{region '#Template'}
	{attribute 'Version' := '1.2.2.0'}
	{attribute 'Tags' := '"LCID": "1031", "Text": "AC, Aggregates, Cooler, Temperature, Controller"'}
	{attribute 'Tags' := '"LCID": "1033", "Text": "AC, Aggregates, Cooler, Temperature, Controller"'}
	{attribute 'Using' := '"Type": "Template", "URI": "BA2_Param"'}
	{attribute 'Using' := '"Type": "Template", "URI": "EC_AMEV"'}
	{attribute 'Description' := '"LCID": "1031", "Text": "Kühler Zuluft Regler Temperatur"'}
	{attribute 'Description' := '"LCID": "1033", "Text": "Cooler Supply air controller temperature"'}
{endregion}
FUNCTION_BLOCK FB_BA_AC_ColTSuACtrl EXTENDS FB_BA_View
VAR_INPUT
	bEn						: BOOL;
	fSpTSuA					: REAL;// Sollwert Temperatur kühlen // Setpoint temperature cooling
	fTSuA					: REAL;// Zuluft Temperatur // Supply air temperature
	bSync					: BOOL;
	fSync					: REAL;
END_VAR
VAR_OUTPUT
	fY              		: REAL;
	bIsActive				: BOOL;	//	active sequence controller
	bOpState				: BOOL;	//	Release sequence link, sequence control is active	
END_VAR
VAR_INPUT CONSTANT
	Ctrl					: FB_BA_LoopSeq;
END_VAR

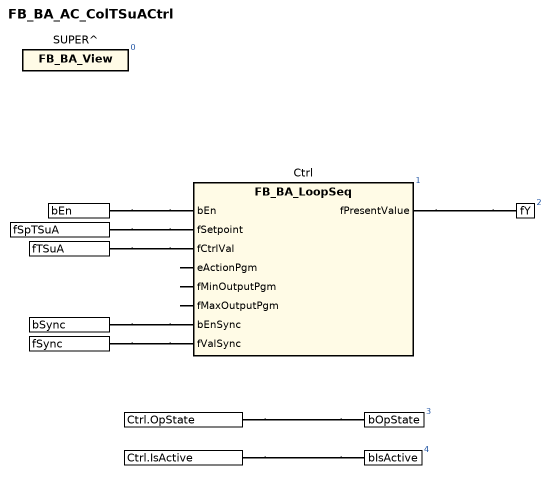
SUPER^(); // FB_BA_View
Ctrl(bEn := bEn, fSetpoint := fSpTSuA, fCtrlVal := fTSuA, bEnSync := bSync, fValSync := fSync); // FB_BA_LoopSeq
fY := Ctrl.fPresentValue;
bOpState := Ctrl.OpState;
bIsActive := Ctrl.IsActive;

METHOD FB_init : BOOL
VAR_INPUT
	bInitRetains : BOOL; // if TRUE, the retain variables are initialized (warm start / cold start)
	bInCopyCode : BOOL;  // if TRUE, the instance afterwards gets moved into the copy code (online change)
END_VAR
Ctrl.iParent						:= THIS^;
Ctrl.iLabel							:= LblCmpAC.Cooler_TSuACtrl_Ctrl; 
Ctrl.sObjectName					:= '{Idx=01}';
Ctrl.eOpMode						:= BA2_Param.nLoop_DefOpMode;								 	 										 
Ctrl.eOutputUnit					:= E_BA_Unit.eOther_Percent;
Ctrl.eActionRm						:= E_BA_Action.eDirect;
Ctrl.fProportionalConstant			:= 3;
Ctrl.fIntegralConstant				:= 180;
Ctrl.fDerivativeConstant			:= 0;
Ctrl.fMaxOutputRm 					:= 100;
Ctrl.fMinOutputRm					:= 0;
Ctrl.fCOVIncrement					:= 0;
Ctrl.nDampConstant					:= 0;
Ctrl.fNeutralZone					:= 0;
END_METHOD

END_FUNCTION_BLOCK

(* stored: Version 1.1.0.1, ProductVersion 3.1.4024.9
   POU FB_BA_AC_ColTSuACtrl: Id {00f77247-410d-4136-a871-d54a2156b99a}, SpecialFunc None
   Method FB_init: Id {d7d20e92-4553-4504-9685-492b4e0687c5} *)
